Yaskawa INFORM job: GAS-OFF.JBI

/JOB
//NAME GAS-OFF
//POS
///NPOS 0,0,0,0,0,0
//INST
///DATE 2015/09/29 09:05
///ATTR SC,RW,MC
NOP
DOUT OT#(51) OFF
TIMER T=0.50
END
